SYSTEM TANK_VIEWL (* Level Control System View+HMI *)
  (* Standard: 61499-1; Classification: Simulation; ApplicationDomain: Process Control *)
  (* Version 0.1, 2004-09-02, JHC, Rockwell Automation, Separated TANK, VALVE, PUMP resources. *)
  (* Version 0.0, 2004-08-20, JHC, Rockwell Automation, Adapted from DRILL_VIEWL *)
  DEVICE HMI : FRAME_DEVICE
    RESOURCE VALVE : PANEL_RESOURCE
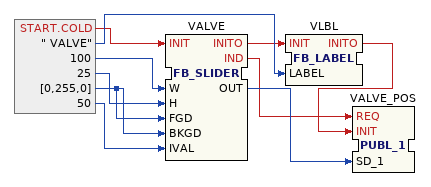
      FBS
        VALVE_POS : PUBL_1;
        VALVE : FB_SLIDER;
        VLBL : FB_LABEL;
      END_FBS
      EVENT_CONNECTIONS
        START.COLD TO VALVE.INIT;
        VALVE.INITO TO VLBL.INIT;
        VALVE.IND TO VALVE_POS.REQ;
        VLBL.INITO TO VALVE_POS.INIT;
      END_CONNECTIONS
      DATA_CONNECTIONS
        VALVE.OUT TO VALVE_POS.SD_1;
        " VALVE" TO VLBL.LABEL;
        100 TO VALVE.W;
        25 TO VALVE.H;
        [0,255,0] TO VALVE.FGD;
        [0,255,0] TO VALVE.BKGD;
        50 TO VALVE.IVAL;
      END_CONNECTIONS
    END_RESOURCE
    RESOURCE TANK : PANEL_RESOURCE
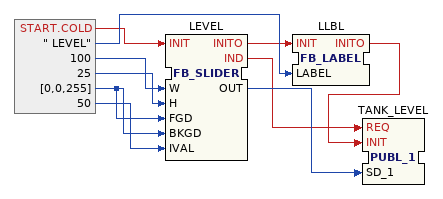
      FBS
        TANK_LEVEL : PUBL_1;
        LEVEL : FB_SLIDER;
        LLBL : FB_LABEL;
      END_FBS
      EVENT_CONNECTIONS
        LEVEL.INITO TO LLBL.INIT;
        LEVEL.IND TO TANK_LEVEL.REQ;
        START.COLD TO LEVEL.INIT;
        LLBL.INITO TO TANK_LEVEL.INIT;
      END_CONNECTIONS
      DATA_CONNECTIONS
        " LEVEL" TO LLBL.LABEL;
        100 TO LEVEL.W;
        25 TO LEVEL.H;
        LEVEL.OUT TO TANK_LEVEL.SD_1;
        [0,0,255] TO LEVEL.FGD;
        [0,0,255] TO LEVEL.BKGD;
        50 TO LEVEL.IVAL;
      END_CONNECTIONS
    END_RESOURCE
    RESOURCE PUMP : PANEL_RESOURCE
      FBS
        PUMP_POS : PUBL_1;
        PUMP : FB_SLIDER;
        PLBL : FB_LABEL;
        PCONV : UNSCALE;
      END_FBS
      EVENT_CONNECTIONS
        PUMP.INITO TO PLBL.INIT;
        PLBL.INITO TO PUMP_POS.INIT;
        PUMP.IND TO PCONV.REQ;
        PCONV.CNF TO PUMP_POS.REQ;
        START.COLD TO PUMP.INIT;
      END_CONNECTIONS
      DATA_CONNECTIONS
        PUMP.OUT TO PCONV.IN;
        " PUMP" TO PLBL.LABEL;
        100 TO PUMP.W;
        25 TO PUMP.H;
        PCONV.OUT TO PUMP_POS.SD_1;
        360 TO PCONV.MAX;
        [255,0,0] TO PUMP.FGD;
        [255,0,0] TO PUMP.BKGD;
        50 TO PUMP.IVAL;
      END_CONNECTIONS
    END_RESOURCE
  END_DEVICE
  DEVICE VIEW : FRAME_DEVICE
    RESOURCE VALVE : VIEW_PANEL
      FBS
        VALVE_POS : SUBL_1;
        VALVE : VALVE_VIEW;
      END_FBS
      EVENT_CONNECTIONS
        START.COLD TO VALVE_POS.INIT;
        VALVE_POS.INITO TO VALVE.INIT;
        VALVE_POS.IND TO VALVE.REQ;
      END_CONNECTIONS
      DATA_CONNECTIONS
        VALVE_POS.RD_1 TO VALVE.POS;
        50 TO VALVE.DIA;
        [0,255,0] TO VALVE.FGD;
      END_CONNECTIONS
    END_RESOURCE
    RESOURCE TANK : VIEW_PANEL
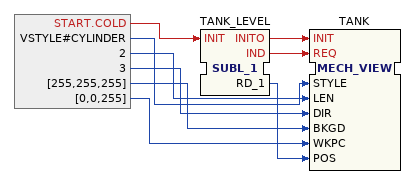
      FBS
        TANK : MECH_VIEW;
        TANK_LEVEL : SUBL_1;
      END_FBS
      EVENT_CONNECTIONS
        TANK_LEVEL.INITO TO TANK.INIT;
        TANK_LEVEL.IND TO TANK.REQ;
        START.COLD TO TANK_LEVEL.INIT;
      END_CONNECTIONS
      DATA_CONNECTIONS
        VSTYLE#CYLINDER TO TANK.STYLE;
        2 TO TANK.LEN;
        3 TO TANK.DIR;
        [255,255,255] TO TANK.BKGD;
        [0,0,255] TO TANK.WKPC;
        TANK_LEVEL.RD_1 TO TANK.POS;
      END_CONNECTIONS
    END_RESOURCE
    RESOURCE PUMP : VIEW_PANEL
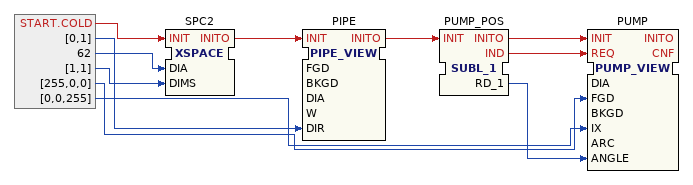
      FBS
        PUMP_POS : SUBL_1;
        SPC2 : XSPACE;
        PIPE : PIPE_VIEW;
        PUMP : PUMP_VIEW;
      END_FBS
      EVENT_CONNECTIONS
        SPC2.INITO TO PIPE.INIT;
        START.COLD TO SPC2.INIT;
        PIPE.INITO TO PUMP_POS.INIT;
        PUMP_POS.INITO TO PUMP.INIT;
        PUMP_POS.IND TO PUMP.REQ;
      END_CONNECTIONS
      DATA_CONNECTIONS
        [0,1] TO PIPE.DIR;
        62 TO SPC2.DIA;
        [1,1] TO SPC2.DIMS;
        PUMP_POS.RD_1 TO PUMP.ANGLE;
        [255,0,0] TO PUMP.FGD;
        [0,0,255] TO PUMP.IX;
      END_CONNECTIONS
    END_RESOURCE
    DATA_CONNECTIONS
      [1,2] TO TANK.SIZE;
      75 TO TANK.DIA;
      50 TO PUMP.DIA;
      [4,1] TO PUMP.SIZE;
      50 TO VALVE.DIA;
      [1,3] TO VALVE.SIZE;
    END_CONNECTIONS
  END_DEVICE
  DATA_CONNECTIONS (* parameter values *)
    [100,100,150,120] TO HMI.BOUNDS;
    [3,1] TO HMI.GRID;
    [250,100,175,250] TO VIEW.BOUNDS;
  END_CONNECTIONS
END_SYSTEM
